Staubli VAL3: CommType.pjx

--- CommType.pjx ---
Parameters version=s7.3 stackSize=5000 millimeterUnit=true
Data file=CommType.dtx

--- CommType.dtx ---
public num nRequest = 2
public num nResponse = 3
